FUNCTION_BLOCK FB_SubsystemCompositionCustomized


(*
fbPACcapacityCounter(sNetId:= '172.31.5.66.1.1', // enter ams net id of IPC
	                 sFileName:='C:\Users\Test2.csv', // enter user file name and path to crate file automatically
                     LogData01:= F_GetTransportControlData(E_FunctionNumber.F_11_001_0200_01_0,1),
	                 LogData02:= F_GetTransportControlData(E_FunctionNumber.F_11_001_0203_01_0,1));
 *)

END_FUNCTION_BLOCK

(* stored: Version 1.1.0.1, ProductVersion 3.1.4024.9
   POU FB_SubsystemCompositionCustomized: Id {087b3c35-0b3c-449d-90dd-291923d8689d}, SpecialFunc None *)
